{attribute 'qualified_only'}
{attribute 'strict'}
{attribute 'to_string'}
TYPE nSealingCorkAssKeyencePN_ErrorCodes :
(
	// Błędy ogólne
	NoError := 0,
	UnKnownAlarm := 53,						// Niezidentyfikowany alarm maszyny
	UnKnownLock := 54,						// Niezidentyfikowana blokada maszyny
	ProgramConfigError := 90,				// Błąd w konfiguracji programu
	
	SensorNotReady:= 193, 
	BadSealingCorkAssembly:= 194, 
	CapNotDetected	:= 197, 
	WrongOringWidth := 196, 
	LackOfOring := 195, 
	CapNotDetectedAndNoOring := 198, 
	WrongOringWidthAndCapNotDetected := 199 
//	CapNotDet:= 173,
//	SealingCapNotDet:= 	
);
END_TYPE

(* stored: Version 1.1.0.1, ProductVersion 3.1.4024.13
   EnumerationTextList nSealingCorkAssKeyencePN_ErrorCodes: Id {87f4e6ec-9f77-49fb-a21c-fd814657599d} *)
